// This function has been automatically generated from the project information.
{attribute 'signature_flag' := '1073741824'}
{attribute 'TcGenerated'}
{attribute 'no-analysis'}
FUNCTION F_GetTitle : WSTRING
VAR_INPUT
	
END_VAR

F_GetTitle := "Tc3PlcTestSuite";

END_FUNCTION

(* stored: Version 1.1.0.1
   POU F_GetTitle: Id {f5776e21-d485-487b-809a-a189afdacb31}, SpecialFunc None *)
